// TIA Portal project "2022.06.06_四则运算万能公式" (V17)

(* hardware
DEVICE "S7-1200 station_1"  S7-1200 Station
   slot 0: "Rack_0"  S7-1200 Rack  Rack  V1.0
   slot 1: "PLC_1"  CPU 1212C DC/DC/DC  6ES7 212-1AE40-0XB0  V4.5
*)

// ===== PLC "PLC_1"  CPU 1212C DC/DC/DC =====

VAR_GLOBAL   // PLC tag table "默认变量表"
   "Tag_2" AT %MW100 : Word;
   "Tag_3" AT %MW102 : UInt;
   "Tag_4" AT %MW104 : UInt;
   "Tag_5" AT %MW106 : UInt;
   "Tag_6" AT %I0.0 : Bool;
   "Tag_7" AT %M0.0 : Bool;
   "X(2)" AT %MW10 : Word;
   "Tag_9" AT %MW12 : UInt;
   "X" AT %MW0 : Word;
   "a" AT %MW2 : Word;
   "b" AT %MW4 : Int;
   "c" AT %MW8 : Int;
   "e" AT %MD0 : Real;
   "Tag_10" AT %MD2 : Real;
   "f" AT %MD4 : Real;
   "g" AT %MD8 : Real;
   "X(1)" AT %MD12 : Real;
   "Tag_8" AT %MD16 : Real;
END_VAR

ORGANIZATION_BLOCK "Main"   // OB1, LAD, ProgramCycle
TITLE = "Main Program Sweep (Cycle)"
{ S7_Optimized_Access := 'TRUE' }
VERSION : 0.1
   VAR_INPUT
      Initial_Call : Bool;   // Initial call of this OB
      Remanence : Bool;   // =True, if remanent data are available
   END_VAR
BEGIN

REGION Network 1
   // Y=2x+6
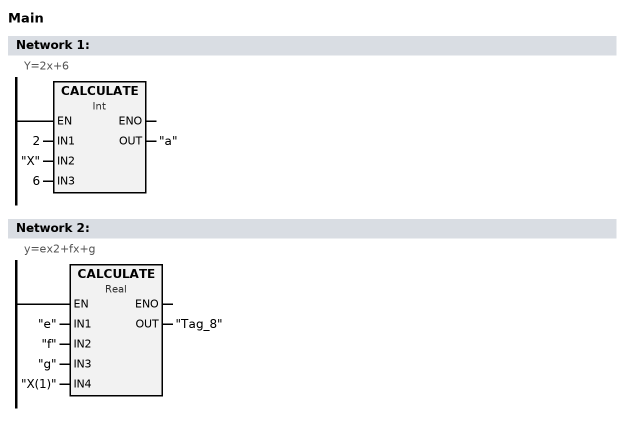
   RUNG wire#powerrail
      { S7_Templates := "SrcType := Int"; S7_Expression := "IN1*IN2+IN3" } Calculate(in1 := 2, in2 := "X", in3 := 6, out => "a")
   END_RUNG
   // the same network as SCL:
   "a" := 2*"X"+6;
END_REGION

REGION Network 2
   // y=ex2+fx+g
   RUNG wire#powerrail
      { S7_Templates := "SrcType := Real"; S7_Expression := "IN1*SQR(IN4)+IN2*IN4+IN3" } Calculate(in1 := "e", in2 := "f", in3 := "g", in4 := "X(1)", out => "Tag_8")
   END_RUNG
   // the same network as SCL:
   "Tag_8" := "e"*SQR("X(1)")+"f"*"X(1)"+"g";
END_REGION
END_ORGANIZATION_BLOCK